FUNCTION_BLOCK FB_ManualControl
VAR_INPUT
	eMode 	: E_Mode;
	eStatus : E_Status;
	stParam : ST_Parameters;
END_VAR
VAR_OUTPUT
	fControlOutputNormalized : LREAL;
END_VAR
VAR
	fbJoystick 			: FB_Joystick; 
	fbOpenLoopControl  	: FB_OpenLoopControl; 
END_VAR

fbJoystick(
	bEnable := (eMode = E_Mode.Manual),
	stParam := stParam,
	fNormalizedInput := G_Work.fJoystickY,
);

fbOpenLoopControl(
	bEnable := (eMode = E_Mode.Manual),
	stParam := stParam,
	fInput_ms := fbJoystick.fOuput,
	fNormalizedOutput => fControlOutputNormalized
);

END_FUNCTION_BLOCK

(* stored: Version 1.1.0.1, ProductVersion 3.1.4024.10
   POU FB_ManualControl: Id {1cb952f3-59ec-4dc1-98d9-dc6242ed003b}, SpecialFunc None *)
